(* CoDeSys 2.3.9.47 project: PUMP SUCCESS.pro *)
(* Libraries: Nexgenie.lib 28.8.18 12:27:24, Standard.lib 28.8.18 12:27:25, Nexgenie_Util.lib 28.8.18 12:27:24, Nexgenie_H.lib 28.8.18 12:27:24, VAW.lib 28.8.18 12:27:25, Modbus.lib 28.8.18 12:27:24 *)

(* PLC configuration (modules and I/O channels)
Nexgenie1000 [Root] node -1, in %IB0 out %QB0
  Nexgenie [Nexgenie] node 0, in %IB0 out %QB0
*)

(* POU PLC_PRG, LD *)
PROGRAM PLC_PRG
VAR
	SB: BOOL;
	APUMP: BOOL;
	STOP1: BOOL;
	STOP2: BOOL;
	BPUMP: BOOL;
	STOP3: BOOL;
	CPUMP: BOOL;
	MAINCONTRACTOR: BOOL;
	ALARM: BOOL;
END_VAR
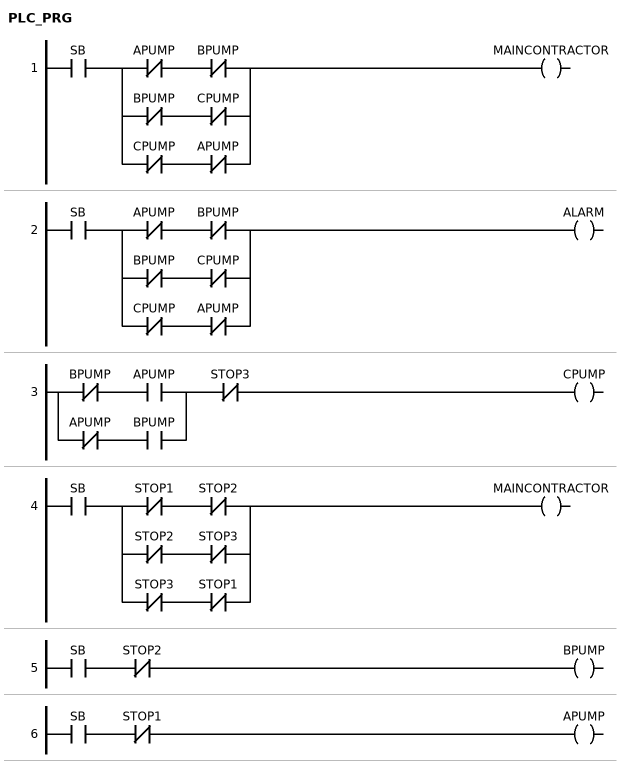
_LD_ (* Ladder Diagram *)
NETWORK 1
	[SB] - { [/APUMP] - [/BPUMP] | [/BPUMP] - [/CPUMP] | [/CPUMP] - [/APUMP] } --- (MAINCONTRACTOR)
NETWORK 2
	[SB] - { [/APUMP] - [/BPUMP] | [/BPUMP] - [/CPUMP] | [/CPUMP] - [/APUMP] } --- (ALARM)
NETWORK 3
	{ [/BPUMP] - [APUMP] | [/APUMP] - [BPUMP] } - [/STOP3] --- (CPUMP)
NETWORK 4
	[SB] - { [/STOP1] - [/STOP2] | [/STOP2] - [/STOP3] | [/STOP3] - [/STOP1] } --- (MAINCONTRACTOR)
NETWORK 5
	[SB] - [/STOP2] --- (BPUMP)
NETWORK 6
	[SB] - [/STOP1] --- (APUMP)
_END_LD_
(* the same logic as Structured Text *)
(* Network 1 *)
MAINCONTRACTOR := SB AND (NOT APUMP AND NOT BPUMP OR NOT BPUMP AND NOT CPUMP OR NOT CPUMP AND NOT APUMP);
(* Network 2 *)
ALARM := SB AND (NOT APUMP AND NOT BPUMP OR NOT BPUMP AND NOT CPUMP OR NOT CPUMP AND NOT APUMP);
(* Network 3 *)
CPUMP := (NOT BPUMP AND APUMP OR NOT APUMP AND BPUMP) AND NOT STOP3;
(* Network 4 *)
MAINCONTRACTOR := SB AND (NOT STOP1 AND NOT STOP2 OR NOT STOP2 AND NOT STOP3 OR NOT STOP3 AND NOT STOP1);
(* Network 5 *)
BPUMP := SB AND NOT STOP2;
(* Network 6 *)
APUMP := SB AND NOT STOP1;
END_PROGRAM

(* Visualisation LOL
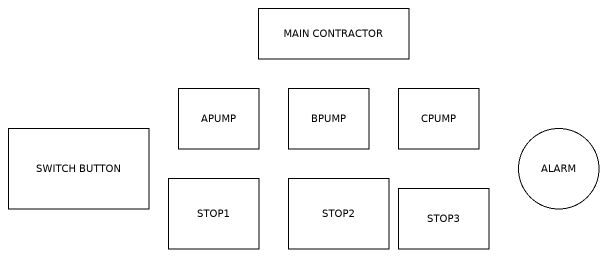
rectangle at (0,160)-(141,241): text "SWITCH BUTTON"; alarm colour if PLC_PRG.SB; toggles PLC_PRG.SB
rounded rectangle at (170,120)-(251,181): text "APUMP"; alarm colour if PLC_PRG.APUMP; toggles PLC_PRG.APUMP
rounded rectangle at (160,210)-(251,281): text "STOP1"; alarm colour if PLC_PRG.STOP1; toggles PLC_PRG.STOP1
rounded rectangle at (280,120)-(361,181): text "BPUMP"; alarm colour if PLC_PRG.BPUMP; toggles PLC_PRG.BPUMP
rounded rectangle at (280,210)-(381,281): text "STOP2"; alarm colour if PLC_PRG.STOP2; toggles PLC_PRG.STOP2
rounded rectangle at (390,120)-(471,181): text "CPUMP"; alarm colour if PLC_PRG.CPUMP; toggles PLC_PRG.CPUMP
rounded rectangle at (390,220)-(481,281): text "STOP3"; alarm colour if PLC_PRG.STOP3; toggles PLC_PRG.STOP3
ellipse at (510,160)-(591,241): text "ALARM"; alarm colour if PLC_PRG.ALARM
rectangle at (250,40)-(401,91): text "MAIN CONTRACTOR"; alarm colour if PLC_PRG.MAINCONTRACTOR; toggles PLC_PRG.MAINCONTRACTOR
*)
